// TIA Portal V18 export
ORGANIZATION_BLOCK "16-Rotunda"   // OB130, LAD, ProgramCycle
TITLE = Rotunda / "Main Program Sweep (Cycle)"
{ S7_Optimized_Access := 'TRUE' }
VERSION : 0.1
// stored: AutoNumber true, IsIECCheckEnabled false, SetENOAutomatically false
   VAR_INPUT
      Initial_Call : Bool;   // Initial call of this OB
      Remanence : Bool;   // =True, if remanent data are available
   END_VAR
   VAR_TEMP
      "Angle Rotunda NormScale" : Real;
   END_VAR
   VAR_TEMP   // added for the SCL form of the ladder/FBD networks
      _w1 : Bool;
      _w2 : Bool;
   END_VAR
BEGIN

REGION Network 1: Rotunda Angle Sensor
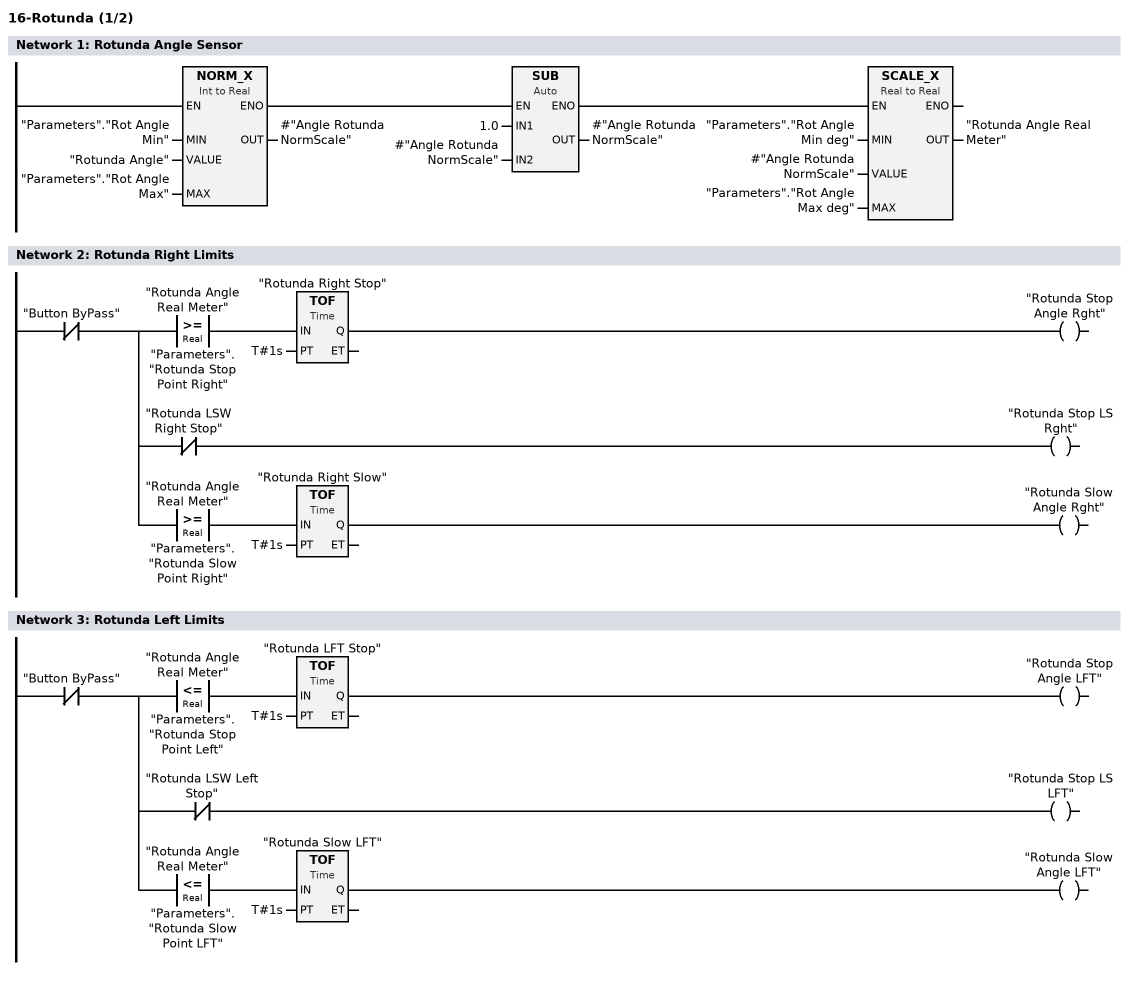
   RUNG wire#powerrail
      { S7_Templates := "[SrcType := Int, DestType := Real]" } Normalize(min := "Parameters"."Rot Angle Min", value := "Rotunda Angle", max := "Parameters"."Rot Angle Max", out => #"Angle Rotunda NormScale")
      Sub(in1 := 1.0, in2 := #"Angle Rotunda NormScale", out => #"Angle Rotunda NormScale")
      { S7_Templates := "[SrcType := Real, DestType := Real]" } Scale(min := "Parameters"."Rot Angle Min deg", value := #"Angle Rotunda NormScale", max := "Parameters"."Rot Angle Max deg", out => "Rotunda Angle Real Meter")
   END_RUNG
   // the same network as SCL:
   #"Angle Rotunda NormScale" := NORM_X(MIN := "Parameters"."Rot Angle Min", VALUE := "Rotunda Angle", MAX := "Parameters"."Rot Angle Max");
   #"Angle Rotunda NormScale" := 1.0 - #"Angle Rotunda NormScale";
   "Rotunda Angle Real Meter" := SCALE_X(MIN := "Parameters"."Rot Angle Min deg", VALUE := #"Angle Rotunda NormScale", MAX := "Parameters"."Rot Angle Max deg");
END_REGION

REGION Network 2: Rotunda Right Limits
   RUNG wire#powerrail
      I_Contact( "Button ByPass" )
      wire#w1
      { S7_Templates := "SrcType := Real" } GE_Contact(in1 := "Rotunda Angle Real Meter", in2 := "Parameters"."Rotunda Stop Point Right")
      { S7_Templates := "time_type := Time" } "Rotunda Right Stop".TOF(pt := T#1s, et =>)
      Coil( "Rotunda Stop Angle Rght" )
   END_RUNG
   RUNG wire#w1
      I_Contact( "Rotunda LSW Right Stop" )
      Coil( "Rotunda Stop LS Rght" )
   END_RUNG
   RUNG wire#w1
      { S7_Templates := "SrcType := Real" } GE_Contact(in1 := "Rotunda Angle Real Meter", in2 := "Parameters"."Rotunda Slow Point Right")
      { S7_Templates := "time_type := Time" } "Rotunda Right Slow".TOF(pt := T#1s, et =>)
      Coil( "Rotunda Slow Angle Rght" )
   END_RUNG
   // the same network as SCL:
   "Rotunda Right Stop".TOF(IN := NOT "Button ByPass" AND ("Rotunda Angle Real Meter" >= "Parameters"."Rotunda Stop Point Right"),
                           PT := T#1s);
   "Rotunda Stop Angle Rght" := "Rotunda Right Stop".Q;
   "Rotunda Stop LS Rght" := NOT "Button ByPass" AND NOT "Rotunda LSW Right Stop";
   "Rotunda Right Slow".TOF(IN := NOT "Button ByPass" AND ("Rotunda Angle Real Meter" >= "Parameters"."Rotunda Slow Point Right"),
                           PT := T#1s);
   "Rotunda Slow Angle Rght" := "Rotunda Right Slow".Q;
END_REGION

REGION Network 3: Rotunda Left Limits
   RUNG wire#powerrail
      I_Contact( "Button ByPass" )
      wire#w1
      { S7_Templates := "SrcType := Real" } LE_Contact(in1 := "Rotunda Angle Real Meter", in2 := "Parameters"."Rotunda Stop Point Left")
      { S7_Templates := "time_type := Time" } "Rotunda LFT Stop".TOF(pt := T#1s, et =>)
      Coil( "Rotunda Stop Angle LFT" )
   END_RUNG
   RUNG wire#w1
      I_Contact( "Rotunda LSW Left Stop" )
      Coil( "Rotunda Stop LS LFT" )
   END_RUNG
   RUNG wire#w1
      { S7_Templates := "SrcType := Real" } LE_Contact(in1 := "Rotunda Angle Real Meter", in2 := "Parameters"."Rotunda Slow Point LFT")
      { S7_Templates := "time_type := Time" } "Rotunda Slow LFT".TOF(pt := T#1s, et =>)
      Coil( "Rotunda Slow Angle LFT" )
   END_RUNG
   // the same network as SCL:
   "Rotunda LFT Stop".TOF(IN := NOT "Button ByPass" AND ("Rotunda Angle Real Meter" <= "Parameters"."Rotunda Stop Point Left"),
                          PT := T#1s);
   "Rotunda Stop Angle LFT" := "Rotunda LFT Stop".Q;
   "Rotunda Stop LS LFT" := NOT "Button ByPass" AND NOT "Rotunda LSW Left Stop";
   "Rotunda Slow LFT".TOF(IN := NOT "Button ByPass" AND ("Rotunda Angle Real Meter" <= "Parameters"."Rotunda Slow Point LFT"),
                          PT := T#1s);
   "Rotunda Slow Angle LFT" := "Rotunda Slow LFT".Q;
END_REGION

REGION Network 4: Rotunda Stop-Slow Limits
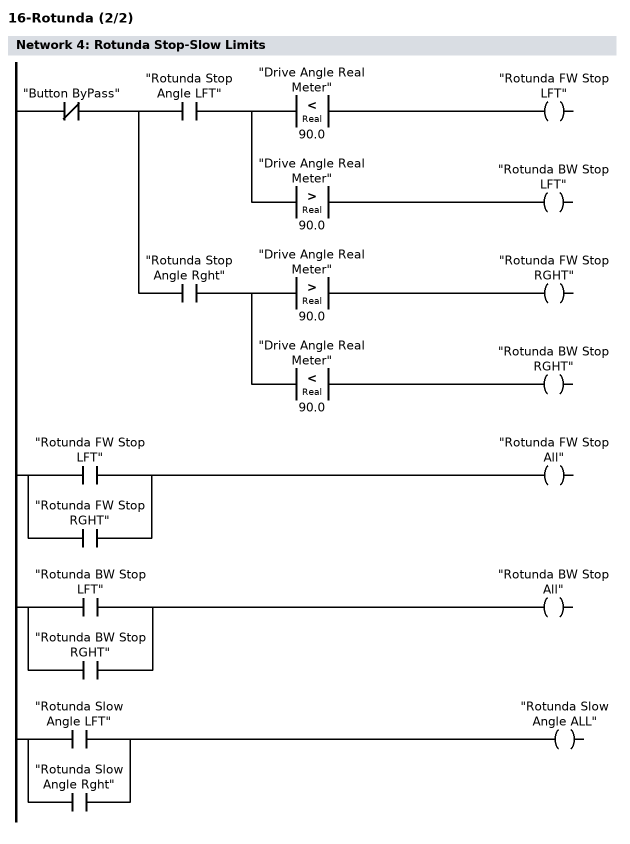
   RUNG wire#powerrail
      I_Contact( "Button ByPass" )
      wire#w1
      Contact( "Rotunda Stop Angle LFT" )
      wire#w2
      { S7_Templates := "SrcType := Real" } LT_Contact(in1 := "Drive Angle Real Meter", in2 := 90.0)
      Coil( "Rotunda FW Stop LFT" )
   END_RUNG
   RUNG wire#w2
      { S7_Templates := "SrcType := Real" } GT_Contact(in1 := "Drive Angle Real Meter", in2 := 90.0)
      Coil( "Rotunda BW Stop LFT" )
   END_RUNG
   RUNG wire#w1
      Contact( "Rotunda Stop Angle Rght" )
      wire#w3
      { S7_Templates := "SrcType := Real" } GT_Contact(in1 := "Drive Angle Real Meter", in2 := 90.0)
      Coil( "Rotunda FW Stop RGHT" )
   END_RUNG
   RUNG wire#w3
      { S7_Templates := "SrcType := Real" } LT_Contact(in1 := "Drive Angle Real Meter", in2 := 90.0)
      Coil( "Rotunda BW Stop RGHT" )
   END_RUNG
   RUNG wire#powerrail
      Contact( "Rotunda FW Stop LFT" )
      wire#w4
      Coil( "Rotunda FW Stop All" )
   END_RUNG
   RUNG wire#powerrail
      Contact( "Rotunda FW Stop RGHT" )
   END_RUNG wire#w4
   RUNG wire#powerrail
      Contact( "Rotunda BW Stop LFT" )
      wire#w5
      Coil( "Rotunda BW Stop All" )
   END_RUNG
   RUNG wire#powerrail
      Contact( "Rotunda BW Stop RGHT" )
   END_RUNG wire#w5
   RUNG wire#powerrail
      Contact( "Rotunda Slow Angle LFT" )
      wire#w6
      Coil( "Rotunda Slow Angle ALL" )
   END_RUNG
   RUNG wire#powerrail
      Contact( "Rotunda Slow Angle Rght" )
   END_RUNG wire#w6
   // the same network as SCL:
   #_w1 := NOT "Button ByPass" AND "Rotunda Stop Angle LFT";
   "Rotunda FW Stop LFT" := #_w1 AND ("Drive Angle Real Meter" < 90.0);
   "Rotunda BW Stop LFT" := #_w1 AND ("Drive Angle Real Meter" > 90.0);
   #_w2 := NOT "Button ByPass" AND "Rotunda Stop Angle Rght";
   "Rotunda FW Stop RGHT" := #_w2 AND ("Drive Angle Real Meter" > 90.0);
   "Rotunda BW Stop RGHT" := #_w2 AND ("Drive Angle Real Meter" < 90.0);
   "Rotunda FW Stop All" := "Rotunda FW Stop LFT" OR "Rotunda FW Stop RGHT";
   "Rotunda BW Stop All" := "Rotunda BW Stop LFT" OR "Rotunda BW Stop RGHT";
   "Rotunda Slow Angle ALL" := "Rotunda Slow Angle LFT" OR "Rotunda Slow Angle Rght";
END_REGION
END_ORGANIZATION_BLOCK
